ABB RobotStudio station: Proyecto_CesarGonzalez.rspag

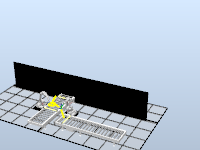
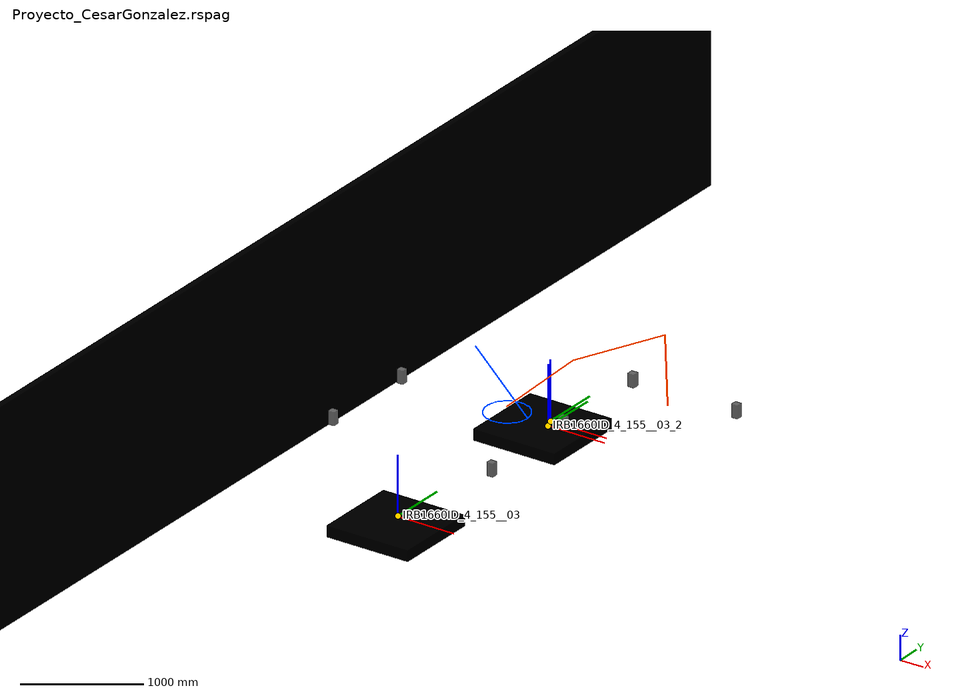
[picture v1: parts stored in the station drawn from their meshes, with robot base, taught points and paths (robot models come from the ABB library and are not in the file)]
--- station ---
Station Proyecto (saved by RobotStudio 21.2.9526.0)
Controller Controlador2, task T_ROB1: task frame (RAPID world) sits at (1630.73, 858.73, 94.26) mm in the station
Controller Controlador1, task T_ROB2: task frame (RAPID world) sits at (1633.69, -1291.95, 100) mm, rotated rx 0 ry 0 rz 90 deg in the station
Controller Controlador1, task T_ROB1: task frame (RAPID world) sits at (1633.69, -1291.95, 100) mm, rotated rx 0 ry 0 rz 90 deg in the station
Controller Controlador1
  mechanical unit ROB_1: IRB1660ID_4_155__03, 6 joints, base frame (0, 0, 0) mm
  mechanical unit ROB_2: IRB1660ID_4_155__03_2, 6 joints, base frame (0, 0, 0) mm
Controller Controlador2
  mechanical unit ROB_1: IRB1660ID_4_155__03_3, 6 joints, base frame (0, 0, 0) mm
Layout (positions relative to the parent item):
  - 950_4000_h2 [part, from Equipment\Conveyor 950 4000 h2.rslib] at (-254.72, -756.17, 0) mm
  - IRB1660ID_4_155__03 [mechanism, from Robots\IRB1660ID_4_155__03.rslib] at (1633.69, -1291.95, 100) mm, rotated rx 0 ry 0 rz 90 deg; joint values [-0.6056, 0.2499, 0.2095, 0.6847, 0.6619, -1.1198] (rad or m)
  - Pedestal1 [part] at (1259.57, -1762.3, 0) mm, size 800 x 800 x 100 mm
  - MyTool [mechanism, from Training Objects\myTool.rslib] at (2186.3, -401.7, 957.93) mm, rotated rx -179.96 ry 39.06 rz -86.55 deg
  - Cubo [part] at (3490.77, -286.76, 436.4) mm, size 400 x 400 x 300 mm
  - Tapa [part] at (2580.97, 4280.73, 447.22) mm, size 400 x 397.8 x 50 mm
  - 950_4000_h2_3 [part, from Equipment\Conveyor 950 4000 h2.rslib] at (3186.02, 749.76, 0) mm, rotated rx 0 ry 0 rz 90 deg
  - Pedestal2 [part] at (1208.56, 374.28, 0) mm, size 800 x 800 x 100 mm
  - IRB1660ID_4_155__03_2 [mechanism, from Robots\IRB1660ID_4_155__03.rslib] at (1674.65, 765.71, 100) mm; joint values [0, 0, 0, 0, 0.5236, 0] (rad or m)
  - PhysicsControl_cinta1 [smart component, from Components\PhysicsControl.rslib]
      properties: Object=cinta1; Behavior=1; SurfaceVelocity=0.2
  - PhysicsControl_cinta2 [smart component, from Components\PhysicsControl.rslib]
      properties: Object=cinta2; Behavior=1; SurfaceVelocity=0.2
  - Source_Cubo [smart component, from Components\Source.rslib]
      properties: Source=Cubo; Copy=(none); Parent=(none); Position=[3.49 -0.286 0.436]; Orientation=[0 0 0]; Transient=true; PhysicsBehavior=3
  - Source_Tapa [smart component, from Components\Source.rslib]
      properties: Source=Tapa; Copy=(none); Parent=(none); Position=[2.68 4.28 0.487]; Orientation=[0 0 0]; Transient=true; PhysicsBehavior=3
  - Pieza_2 [part] at (600.26, 166.12, 428.71) mm, size 60 x 60 x 120 mm
  - Pieza_3 [part] at (598.1, -796.46, 441.5) mm, size 60 x 60 x 120 mm
  - LineSensor_tapa [smart component, from Components\LineSensor.rslib] at (0, 259.06, -11.33) mm
      properties: Start=[2.263156 0.947069 0.47]; End=[3.181577 0.953591 0.47]; Radius=0; SensedPart=(none); SensedPoint=[2.49121630859375 1.20774780273438 0.458671112060547]
    - _sensorPart_ [part], size 918.4 x 6.5 x 0 mm
  - Pieza_4 [part] at (3189.53, 1175.28, 439.43) mm, size 60 x 60 x 120 mm
  - Pieza_5 [part] at (2172.87, 1169.42, 434.14) mm, size 60 x 60 x 120 mm
  - LineSensor_pegamento [smart component, from Components\LineSensor.rslib]
      properties: Start=[2.212913 -0.75684 0.495656]; End=[2.208882 0.177208 0.496891]; Radius=0; SensedPart=(none); SensedPoint=[0 0 0]
    - _sensorPart_ [part], size 4 x 934 x 1.2 mm
  - Pieza_6 [part] at (2178.88, 187.93, 436.89) mm, size 60 x 60 x 120 mm
  - Pieza_7 [part] at (2182.91, -828.74, 435.66) mm, size 60 x 60 x 120 mm
  - LineSensor_final [smart component, from Components\LineSensor.rslib]
      properties: Start=[0.628097 -0.720379 0.5015]; End=[0.630264 0.156269 0.488715]; Radius=0; SensedPart=(none); SensedPoint=[0 0 0]
    - _sensorPart_ [part], size 2.2 x 876.6 x 12.8 mm
  - cinta2 [part] at (2230.42, 4806.6, 338.68) mm, rotated rx 0 ry 0 rz -89.73 deg, size 4000 x 910 x 80 mm
  - cinta1 [part] at (-131.25, -752.86, 358) mm, size 4000 x 910 x 80 mm
  - IRB1660ID_4_155__03_3 [mechanism, from Robots\IRB1660ID_4_155__03.rslib] at (1630.73, 858.73, 94.26) mm; joint values [0, 0, 0, 0, 0.5236, 0] (rad or m)
  - Attacher [smart component, from Components\Attacher.rslib]
      properties: Parent=MyTool_2; Flange=0; Child=(none); Mount=false; Offset=[0 0 0]; Orientation=[0 0 0]
  - Detacher [smart component, from Components\Detacher.rslib]
      properties: Child=(none); KeepPosition=true
  - MyTool_2 [mechanism, from Training Objects\myTool.rslib] at (2575.61, 858.73, 1323.26) mm, rotated rx -180 ry 60 rz -180 deg
  - SimulationEvents [smart component, from Components\SimulationEvents.rslib]
  - Pared [part] at (28.4, -4684.22, 0) mm, size 60 x 10000 x 2000 mm
Attachment: Pedestal1 is attached to IRB1660ID_4_155__03 / Base
Attachment: MyTool is attached to IRB1660ID_4_155__03 / Link6
Attachment: Pedestal2 is attached to IRB1660ID_4_155__03_2 / Base
Attachment: PhysicsControl_cinta2 is attached to 950_4000_h2
Attachment: MyTool_2 is attached to IRB1660ID_4_155__03_3 / Link6
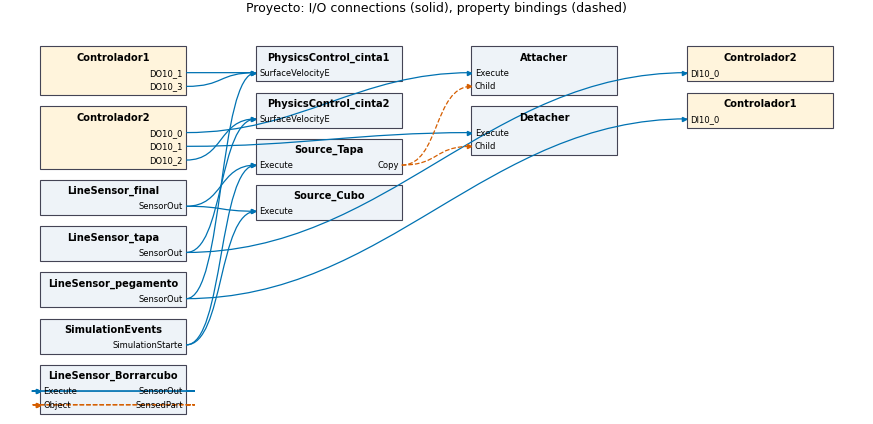
Station logic (signal -> signal, property => property):
  Controlador1.DO10_1 -> PhysicsControl_cinta1.SurfaceVelocityEnabled
  Controlador2.DO10_0 -> Attacher.Execute
  Controlador2.DO10_1 -> Detacher.Execute
  LineSensor_final.SensorOut -> Source_Tapa.Execute
  LineSensor_final.SensorOut -> Source_Cubo.Execute
  LineSensor_tapa.SensorOut -> PhysicsControl_cinta2.SurfaceVelocityEnabled
  LineSensor_pegamento.SensorOut -> PhysicsControl_cinta1.SurfaceVelocityEnabled
  LineSensor_pegamento.SensorOut -> Controlador1.DI10_0
  LineSensor_tapa.SensorOut -> Controlador2.DI10_0
  Controlador1.DO10_3 -> PhysicsControl_cinta1.SurfaceVelocityEnabled
  Controlador2.DO10_2 -> PhysicsControl_cinta2.SurfaceVelocityEnabled
  SimulationEvents.SimulationStarted -> Source_Tapa.Execute
  SimulationEvents.SimulationStarted -> Source_Cubo.Execute
  LineSensor_Borrarcubo.SensorOut -> Sink.Execute
  LineSensor_borrartapa.SensorOut -> Sink_3.Execute
  Source_Tapa.Copy => Detacher.Child
  Source_Tapa.Copy => Attacher.Child
  LineSensor_Borrarcubo.SensedPart => Sink.Object
  LineSensor_borrartapa.SensedPart => Sink_3.Object

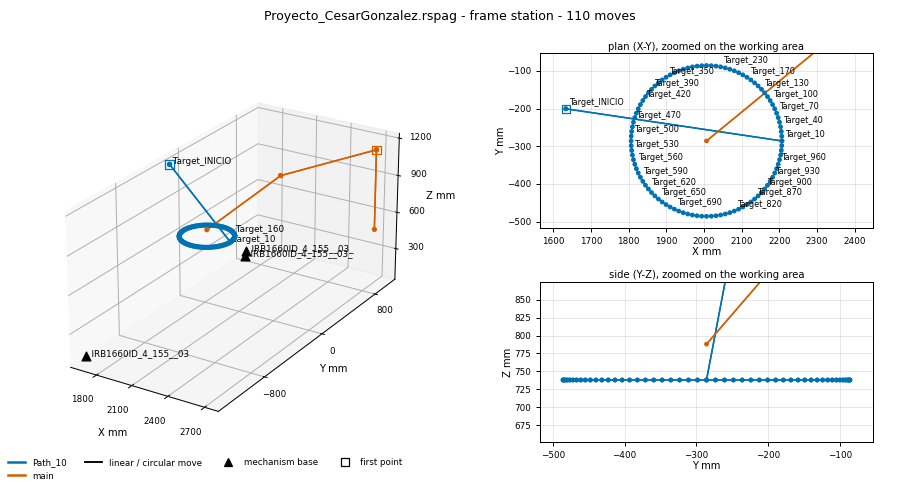
[picture p0: tool path of Proyecto_CesarGonzalez.rspag in frame station, 110 of 110 moves have a stored position in this frame; points joined in program order, loops and branches not executed]
--- Backups/Controlador1/RAPID/TASK1/PROGMOD/CalibData.mod ---
MODULE CalibData
    PERS tooldata MyTool:=[TRUE,[[31.7926,0,229.639],[0.945519,0,0.325568,0]],[1,[0,0,1],[1,0,0,0],0,0,0]];
ENDMODULE

--- Backups/Controlador1/RAPID/TASK1/PROGMOD/Module1.mod ---
MODULE Module1
    CONST robtarget Target_INICIO:=[[1091.194537048,0.000070456,1086.647618205],[0.190809199,-0.000000035,0.981627144,0.000000002],[0,-1,-1,0],[9E+09,9E+09,9E+09,9E+09,9E+09,9E+09]];
    CONST robtarget Target_10:=[[1005.945636056,-573.112362288,637.998901716],[0,-0.031410791,0.999506559,0],[0,0,0,0],[9E+09,9E+09,9E+09,9E+09,9E+09,9E+09]];
    CONST robtarget Target_20:=[[1018.503739937,-572.717707184,637.998901716],[0,-0.031410791,0.999506559,0],[0,0,0,0],[9E+09,9E+09,9E+09,9E+09,9E+09,9E+09]];
    CONST robtarget Target_30:=[[1031.01228267,-571.535300974,637.998901716],[0,-0.031410791,0.999506559,0],[0,0,0,0],[9E+09,9E+09,9E+09,9E+09,9E+09,9E+09]];
    CONST robtarget Target_40:=[[1043.421898751,-569.569810077,637.998901716],[0,-0.031410791,0.999506559,0],[0,0,0,0],[9E+09,9E+09,9E+09,9E+09,9E+09,9E+09]];
    CONST robtarget Target_50:=[[1055.683613094,-566.828991386,637.998901716],[0,-0.031410791,0.999506559,0],[0,0,0,0],[9E+09,9E+09,9E+09,9E+09,9E+09,9E+09]];
    CONST robtarget Target_60:=[[1067.749034316,-563.323661661,637.998901716],[0,-0.031410791,0.999506559,0],[0,0,0,0],[9E+09,9E+09,9E+09,9E+09,9E+09,9E+09]];
    CONST robtarget Target_70:=[[1079.57054571,-559.067654836,637.998901716],[0,-0.031410791,0.999506559,0],[0,0,0,0],[9E+09,9E+09,9E+09,9E+09,9E+09,9E+09]];
    CONST robtarget Target_80:=[[1091.101493172,-554.077767426,637.998901716],[0,-0.031410791,0.999506559,0],[0,0,0,0],[9E+09,9E+09,9E+09,9E+09,9E+09,9E+09]];
    CONST robtarget Target_90:=[[1102.296369321,-548.373692238,637.998901716],[0,-0.031410791,0.999506559,0],[0,0,0,0],[9E+09,9E+09,9E+09,9E+09,9E+09,9E+09]];
    CONST robtarget Target_100:=[[1113.110993094,-541.97794065,637.998901716],[0,-0.031410791,0.999506559,0],[0,0,0,0],[9E+09,9E+09,9E+09,9E+09,9E+09,9E+09]];
    CONST robtarget Target_110:=[[1123.502684113,-534.915753771,637.998901716],[0,-0.031410791,0.999506559,0],[0,0,0,0],[9E+09,9E+09,9E+09,9E+09,9E+09,9E+09]];
    CONST robtarget Target_120:=[[1133.43043112,-527.215002827,637.998901716],[0,-0.031410791,0.999506559,0],[0,0,0,0],[9E+09,9E+09,9E+09,9E+09,9E+09,9E+09]];
    CONST robtarget Target_130:=[[1142.855053833,-518.906079163,637.998901716],[0,-0.031410791,0.999506559,0],[0,0,0,0],[9E+09,9E+09,9E+09,9E+09,9E+09,9E+09]];
    CONST robtarget Target_140:=[[1151.739357573,-510.021774306,637.998901716],[0,-0.031410791,0.999506559,0],[0,0,0,0],[9E+09,9E+09,9E+09,9E+09,9E+09,9E+09]];
    CONST robtarget Target_150:=[[1160.048280052,-500.597150548,637.998901716],[0,-0.031410791,0.999506559,0],[0,0,0,0],[9E+09,9E+09,9E+09,9E+09,9E+09,9E+09]];
    CONST robtarget Target_160:=[[1167.749029747,-490.669402572,637.998901716],[0,-0.031410791,0.999506559,0],[0,0,0,0],[9E+09,9E+09,9E+09,9E+09,9E+09,9E+09]];
    CONST robtarget Target_170:=[[1174.811215319,-480.277710665,637.998901716],[0,-0.031410791,0.999506559,0],[0,0,0,0],[9E+09,9E+09,9E+09,9E+09,9E+09,9E+09]];
    CONST robtarget Target_180:=[[1181.206965548,-469.463086088,637.998901716],[0,-0.031410791,0.999506559,0],[0,0,0,0],[9E+09,9E+09,9E+09,9E+09,9E+09,9E+09]];
    CONST robtarget Target_190:=[[1186.911039328,-458.268209222,637.998901716],[0,-0.031410791,0.999506559,0],[0,0,0,0],[9E+09,9E+09,9E+09,9E+09,9E+09,9E+09]];
    CONST robtarget Target_200:=[[1191.900925287,-446.737261132,637.998901716],[0,-0.031410791,0.999506559,0],[0,0,0,0],[9E+09,9E+09,9E+09,9E+09,9E+09,9E+09]];
    CONST robtarget Target_210:=[[1196.156930626,-434.915749202,637.998901716],[0,-0.031410791,0.999506559,0],[0,0,0,0],[9E+09,9E+09,9E+09,9E+09,9E+09,9E+09]];
    CONST robtarget Target_220:=[[1199.662258834,-422.85032754,637.998901716],[0,-0.031410791,0.999506559,0],[0,0,0,0],[9E+09,9E+09,9E+09,9E+09,9E+09,9E+09]];
    CONST robtarget Target_230:=[[1202.403075983,-410.588612852,637.998901716],[0,-0.031410791,0.999506559,0],[0,0,0,0],[9E+09,9E+09,9E+09,9E+09,9E+09,9E+09]];
    CONST robtarget Target_240:=[[1204.368565319,-398.178996524,637.998901716],[0,-0.031410791,0.999506559,0],[0,0,0,0],[9E+09,9E+09,9E+09,9E+09,9E+09,9E+09]];
    CONST robtarget Target_250:=[[1205.550969956,-385.670453643,637.998901716],[0,-0.031410791,0.999506559,0],[0,0,0,0],[9E+09,9E+09,9E+09,9E+09,9E+09,9E+09]];
    CONST robtarget Target_260:=[[1205.94562348,-373.112349712,637.998901716],[0,-0.031410791,0.999506559,0],[0,0,0,0],[9E+09,9E+09,9E+09,9E+09,9E+09,9E+09]];
    CONST robtarget Target_270:=[[1205.550968376,-360.554245831,637.998901716],[0,-0.031410791,0.999506559,0],[0,0,0,0],[9E+09,9E+09,9E+09,9E+09,9E+09,9E+09]];
    CONST robtarget Target_280:=[[1204.368562167,-348.045703098,637.998901716],[0,-0.031410791,0.999506559,0],[0,0,0,0],[9E+09,9E+09,9E+09,9E+09,9E+09,9E+09]];
    CONST robtarget Target_290:=[[1202.40307127,-335.636087018,637.998901716],[0,-0.031410791,0.999506559,0],[0,0,0,0],[9E+09,9E+09,9E+09,9E+09,9E+09,9E+09]];
    CONST robtarget Target_300:=[[1199.662252579,-323.374372674,637.998901716],[0,-0.031410791,0.999506559,0],[0,0,0,0],[9E+09,9E+09,9E+09,9E+09,9E+09,9E+09]];
    CONST robtarget Target_310:=[[1196.156922853,-311.308951453,637.998901716],[0,-0.031410791,0.999506559,0],[0,0,0,0],[9E+09,9E+09,9E+09,9E+09,9E+09,9E+09]];
    CONST robtarget Target_320:=[[1191.900916029,-299.487440058,637.998901716],[0,-0.031410791,0.999506559,0],[0,0,0,0],[9E+09,9E+09,9E+09,9E+09,9E+09,9E+09]];
    CONST robtarget Target_330:=[[1186.911028619,-287.956492596,637.998901716],[0,-0.031410791,0.999506559,0],[0,0,0,0],[9E+09,9E+09,9E+09,9E+09,9E+09,9E+09]];
    CONST robtarget Target_340:=[[1181.206953431,-276.761616447,637.998901716],[0,-0.031410791,0.999506559,0],[0,0,0,0],[9E+09,9E+09,9E+09,9E+09,9E+09,9E+09]];
    CONST robtarget Target_350:=[[1174.811201842,-265.946992674,637.998901716],[0,-0.031410791,0.999506559,0],[0,0,0,0],[9E+09,9E+09,9E+09,9E+09,9E+09,9E+09]];
    CONST robtarget Target_360:=[[1167.749014963,-255.555301655,637.998901716],[0,-0.031410791,0.999506559,0],[0,0,0,0],[9E+09,9E+09,9E+09,9E+09,9E+09,9E+09]];
    CONST robtarget Target_370:=[[1160.048264019,-245.627554648,637.998901716],[0,-0.031410791,0.999506559,0],[0,0,0,0],[9E+09,9E+09,9E+09,9E+09,9E+09,9E+09]];
    CONST robtarget Target_380:=[[1151.739340356,-236.202931935,637.998901716],[0,-0.031410791,0.999506559,0],[0,0,0,0],[9E+09,9E+09,9E+09,9E+09,9E+09,9E+09]];
    CONST robtarget Target_390:=[[1142.855035499,-227.318628195,637.998901716],[0,-0.031410791,0.999506559,0],[0,0,0,0],[9E+09,9E+09,9E+09,9E+09,9E+09,9E+09]];
    CONST robtarget Target_400:=[[1133.43041174,-219.009705717,637.998901716],[0,-0.031410791,0.999506559,0],[0,0,0,0],[9E+09,9E+09,9E+09,9E+09,9E+09,9E+09]];
    CONST robtarget Target_410:=[[1123.502663765,-211.308956021,637.998901716],[0,-0.031410791,0.999506559,0],[0,0,0,0],[9E+09,9E+09,9E+09,9E+09,9E+09,9E+09]];
    CONST robtarget Target_420:=[[1113.110971858,-204.246770449,637.998901716],[0,-0.031410791,0.999506559,0],[0,0,0,0],[9E+09,9E+09,9E+09,9E+09,9E+09,9E+09]];
    CONST robtarget Target_430:=[[1102.29634728,-197.851020221,637.998901716],[0,-0.031410791,0.999506559,0],[0,0,0,0],[9E+09,9E+09,9E+09,9E+09,9E+09,9E+09]];
    CONST robtarget Target_440:=[[1091.101470414,-192.14694644,637.998901716],[0,-0.031410791,0.999506559,0],[0,0,0,0],[9E+09,9E+09,9E+09,9E+09,9E+09,9E+09]];
    CONST robtarget Target_450:=[[1079.570522325,-187.157060481,637.998901716],[0,-0.031410791,0.999506559,0],[0,0,0,0],[9E+09,9E+09,9E+09,9E+09,9E+09,9E+09]];
    CONST robtarget Target_460:=[[1067.749010395,-182.901055143,637.998901716],[0,-0.031410791,0.999506559,0],[0,0,0,0],[9E+09,9E+09,9E+09,9E+09,9E+09,9E+09]];
    CONST robtarget Target_470:=[[1055.683588733,-179.395726935,637.998901716],[0,-0.031410791,0.999506559,0],[0,0,0,0],[9E+09,9E+09,9E+09,9E+09,9E+09,9E+09]];
    CONST robtarget Target_480:=[[1043.421874044,-176.654909786,637.998901716],[0,-0.031410791,0.999506559,0],[0,0,0,0],[9E+09,9E+09,9E+09,9E+09,9E+09,9E+09]];
    CONST robtarget Target_490:=[[1031.012257717,-174.689420449,637.998901716],[0,-0.031410791,0.999506559,0],[0,0,0,0],[9E+09,9E+09,9E+09,9E+09,9E+09,9E+09]];
    CONST robtarget Target_500:=[[1018.503714835,-173.507015812,637.998901716],[0,-0.031410791,0.999506559,0],[0,0,0,0],[9E+09,9E+09,9E+09,9E+09,9E+09,9E+09]];
    CONST robtarget Target_510:=[[1005.945610905,-173.112362288,637.998901716],[0,-0.031410791,0.999506559,0],[0,0,0,0],[9E+09,9E+09,9E+09,9E+09,9E+09,9E+09]];
    CONST robtarget Target_520:=[[993.387507024,-173.507017392,637.998901716],[0,-0.031410791,0.999506559,0],[0,0,0,0],[9E+09,9E+09,9E+09,9E+09,9E+09,9E+09]];
    CONST robtarget Target_530:=[[980.878964291,-174.689423601,637.998901716],[0,-0.031410791,0.999506559,0],[0,0,0,0],[9E+09,9E+09,9E+09,9E+09,9E+09,9E+09]];
    CONST robtarget Target_540:=[[968.46934821,-176.654914498,637.998901716],[0,-0.031410791,0.999506559,0],[0,0,0,0],[9E+09,9E+09,9E+09,9E+09,9E+09,9E+09]];
    CONST robtarget Target_550:=[[956.207633867,-179.39573319,637.998901716],[0,-0.031410791,0.999506559,0],[0,0,0,0],[9E+09,9E+09,9E+09,9E+09,9E+09,9E+09]];
    CONST robtarget Target_560:=[[944.142212645,-182.901062915,637.998901716],[0,-0.031410791,0.999506559,0],[0,0,0,0],[9E+09,9E+09,9E+09,9E+09,9E+09,9E+09]];
    CONST robtarget Target_570:=[[932.320701251,-187.15706974,637.998901716],[0,-0.031410791,0.999506559,0],[0,0,0,0],[9E+09,9E+09,9E+09,9E+09,9E+09,9E+09]];
    CONST robtarget Target_580:=[[920.789753788,-192.146957149,637.998901716],[0,-0.031410791,0.999506559,0],[0,0,0,0],[9E+09,9E+09,9E+09,9E+09,9E+09,9E+09]];
    CONST robtarget Target_590:=[[909.59487764,-197.851032337,637.998901716],[0,-0.031410791,0.999506559,0],[0,0,0,0],[9E+09,9E+09,9E+09,9E+09,9E+09,9E+09]];
    CONST robtarget Target_600:=[[898.780253866,-204.246783926,637.998901716],[0,-0.031410791,0.999506559,0],[0,0,0,0],[9E+09,9E+09,9E+09,9E+09,9E+09,9E+09]];
    CONST robtarget Target_610:=[[888.388562848,-211.308970805,637.998901716],[0,-0.031410791,0.999506559,0],[0,0,0,0],[9E+09,9E+09,9E+09,9E+09,9E+09,9E+09]];
    CONST robtarget Target_620:=[[878.460815841,-219.009721749,637.998901716],[0,-0.031410791,0.999506559,0],[0,0,0,0],[9E+09,9E+09,9E+09,9E+09,9E+09,9E+09]];
    CONST robtarget Target_630:=[[869.036193127,-227.318645412,637.998901716],[0,-0.031410791,0.999506559,0],[0,0,0,0],[9E+09,9E+09,9E+09,9E+09,9E+09,9E+09]];
    CONST robtarget Target_640:=[[860.151889387,-236.202950269,637.998901716],[0,-0.031410791,0.999506559,0],[0,0,0,0],[9E+09,9E+09,9E+09,9E+09,9E+09,9E+09]];
    CONST robtarget Target_650:=[[851.842966909,-245.627574028,637.998901716],[0,-0.031410791,0.999506559,0],[0,0,0,0],[9E+09,9E+09,9E+09,9E+09,9E+09,9E+09]];
    CONST robtarget Target_660:=[[844.142217214,-255.555322003,637.998901716],[0,-0.031410791,0.999506559,0],[0,0,0,0],[9E+09,9E+09,9E+09,9E+09,9E+09,9E+09]];
    CONST robtarget Target_670:=[[837.080031642,-265.94701391,637.998901716],[0,-0.031410791,0.999506559,0],[0,0,0,0],[9E+09,9E+09,9E+09,9E+09,9E+09,9E+09]];
    CONST robtarget Target_680:=[[830.684281413,-276.761638488,637.998901716],[0,-0.031410791,0.999506559,0],[0,0,0,0],[9E+09,9E+09,9E+09,9E+09,9E+09,9E+09]];
    CONST robtarget Target_690:=[[824.980207633,-287.956515354,637.998901716],[0,-0.031410791,0.999506559,0],[0,0,0,0],[9E+09,9E+09,9E+09,9E+09,9E+09,9E+09]];
    CONST robtarget Target_700:=[[819.990321673,-299.487463443,637.998901716],[0,-0.031410791,0.999506559,0],[0,0,0,0],[9E+09,9E+09,9E+09,9E+09,9E+09,9E+09]];
    CONST robtarget Target_710:=[[815.734316335,-311.308975373,637.998901716],[0,-0.031410791,0.999506559,0],[0,0,0,0],[9E+09,9E+09,9E+09,9E+09,9E+09,9E+09]];
    CONST robtarget Target_720:=[[812.228988127,-323.374397035,637.998901716],[0,-0.031410791,0.999506559,0],[0,0,0,0],[9E+09,9E+09,9E+09,9E+09,9E+09,9E+09]];
    CONST robtarget Target_730:=[[809.488170978,-335.636111724,637.998901716],[0,-0.031410791,0.999506559,0],[0,0,0,0],[9E+09,9E+09,9E+09,9E+09,9E+09,9E+09]];
    CONST robtarget Target_740:=[[807.522681641,-348.045728052,637.998901716],[0,-0.031410791,0.999506559,0],[0,0,0,0],[9E+09,9E+09,9E+09,9E+09,9E+09,9E+09]];
    CONST robtarget Target_750:=[[806.340277005,-360.554270933,637.998901716],[0,-0.031410791,0.999506559,0],[0,0,0,0],[9E+09,9E+09,9E+09,9E+09,9E+09,9E+09]];
    CONST robtarget Target_760:=[[805.94562348,-373.112374864,637.998901716],[0,-0.031410791,0.999506559,0],[0,0,0,0],[9E+09,9E+09,9E+09,9E+09,9E+09,9E+09]];
    CONST robtarget Target_770:=[[806.340278584,-385.670478745,637.998901716],[0,-0.031410791,0.999506559,0],[0,0,0,0],[9E+09,9E+09,9E+09,9E+09,9E+09,9E+09]];
    CONST robtarget Target_780:=[[807.522684794,-398.179021477,637.998901716],[0,-0.031410791,0.999506559,0],[0,0,0,0],[9E+09,9E+09,9E+09,9E+09,9E+09,9E+09]];
    CONST robtarget Target_790:=[[809.488175691,-410.588637558,637.998901716],[0,-0.031410791,0.999506559,0],[0,0,0,0],[9E+09,9E+09,9E+09,9E+09,9E+09,9E+09]];
    CONST robtarget Target_800:=[[812.228994382,-422.850351901,637.998901716],[0,-0.031410791,0.999506559,0],[0,0,0,0],[9E+09,9E+09,9E+09,9E+09,9E+09,9E+09]];
    CONST robtarget Target_810:=[[815.734324107,-434.915773123,637.998901716],[0,-0.031410791,0.999506559,0],[0,0,0,0],[9E+09,9E+09,9E+09,9E+09,9E+09,9E+09]];
    CONST robtarget Target_820:=[[819.990330932,-446.737284517,637.998901716],[0,-0.031410791,0.999506559,0],[0,0,0,0],[9E+09,9E+09,9E+09,9E+09,9E+09,9E+09]];
    CONST robtarget Target_830:=[[824.980218342,-458.26823198,637.998901716],[0,-0.031410791,0.999506559,0],[0,0,0,0],[9E+09,9E+09,9E+09,9E+09,9E+09,9E+09]];
    CONST robtarget Target_840:=[[830.68429353,-469.463108128,637.998901716],[0,-0.031410791,0.999506559,0],[0,0,0,0],[9E+09,9E+09,9E+09,9E+09,9E+09,9E+09]];
    CONST robtarget Target_850:=[[837.080045118,-480.277731902,637.998901716],[0,-0.031410791,0.999506559,0],[0,0,0,0],[9E+09,9E+09,9E+09,9E+09,9E+09,9E+09]];
    CONST robtarget Target_860:=[[844.142231997,-490.66942292,637.998901716],[0,-0.031410791,0.999506559,0],[0,0,0,0],[9E+09,9E+09,9E+09,9E+09,9E+09,9E+09]];
    CONST robtarget Target_870:=[[851.842982941,-500.597169927,637.998901716],[0,-0.031410791,0.999506559,0],[0,0,0,0],[9E+09,9E+09,9E+09,9E+09,9E+09,9E+09]];
    CONST robtarget Target_880:=[[860.151906605,-510.021792641,637.998901716],[0,-0.031410791,0.999506559,0],[0,0,0,0],[9E+09,9E+09,9E+09,9E+09,9E+09,9E+09]];
    CONST robtarget Target_890:=[[869.036211462,-518.906096381,637.998901716],[0,-0.031410791,0.999506559,0],[0,0,0,0],[9E+09,9E+09,9E+09,9E+09,9E+09,9E+09]];
    CONST robtarget Target_900:=[[878.46083522,-527.215018859,637.998901716],[0,-0.031410791,0.999506559,0],[0,0,0,0],[9E+09,9E+09,9E+09,9E+09,9E+09,9E+09]];
    CONST robtarget Target_910:=[[888.388583196,-534.915768555,637.998901716],[0,-0.031410791,0.999506559,0],[0,0,0,0],[9E+09,9E+09,9E+09,9E+09,9E+09,9E+09]];
    CONST robtarget Target_920:=[[898.780275103,-541.977954127,637.998901716],[0,-0.031410791,0.999506559,0],[0,0,0,0],[9E+09,9E+09,9E+09,9E+09,9E+09,9E+09]];
    CONST robtarget Target_930:=[[909.59489968,-548.373704355,637.998901716],[0,-0.031410791,0.999506559,0],[0,0,0,0],[9E+09,9E+09,9E+09,9E+09,9E+09,9E+09]];
    CONST robtarget Target_940:=[[920.789776546,-554.077778135,637.998901716],[0,-0.031410791,0.999506559,0],[0,0,0,0],[9E+09,9E+09,9E+09,9E+09,9E+09,9E+09]];
    CONST robtarget Target_950:=[[932.320724636,-559.067664095,637.998901716],[0,-0.031410791,0.999506559,0],[0,0,0,0],[9E+09,9E+09,9E+09,9E+09,9E+09,9E+09]];
    CONST robtarget Target_960:=[[944.142236566,-563.323669433,637.998901716],[0,-0.031410791,0.999506559,0],[0,0,0,0],[9E+09,9E+09,9E+09,9E+09,9E+09,9E+09]];
    CONST robtarget Target_970:=[[956.207658228,-566.828997641,637.998901716],[0,-0.031410791,0.999506559,0],[0,0,0,0],[9E+09,9E+09,9E+09,9E+09,9E+09,9E+09]];
    CONST robtarget Target_980:=[[968.469372916,-569.56981479,637.998901716],[0,-0.031410791,0.999506559,0],[0,0,0,0],[9E+09,9E+09,9E+09,9E+09,9E+09,9E+09]];
    CONST robtarget Target_990:=[[980.878989244,-571.535304127,637.998901716],[0,-0.031410791,0.999506559,0],[0,0,0,0],[9E+09,9E+09,9E+09,9E+09,9E+09,9E+09]];
    CONST robtarget Target_1000:=[[993.387532125,-572.717708763,637.998901716],[0,-0.031410791,0.999506559,0],[0,0,0,0],[9E+09,9E+09,9E+09,9E+09,9E+09,9E+09]];
    CONST robtarget Target_1010:=[[1005.945636056,-573.112362288,637.998901716],[0,-0.031410791,0.999506559,0],[0,0,0,0],[9E+09,9E+09,9E+09,9E+09,9E+09,9E+09]];

    PROC Path_10()

        MoveL Target_INICIO,v1000,z100,MyTool\WObj:=wobj0;
        MoveL Target_10,v1000,z100,MyTool\WObj:=wobj0;
        MoveL Target_20,v1000,z100,MyTool\WObj:=wobj0;
        MoveL Target_30,v1000,z100,MyTool\WObj:=wobj0;
        MoveL Target_40,v1000,z100,MyTool\WObj:=wobj0;
        MoveL Target_50,v1000,z100,MyTool\WObj:=wobj0;
        MoveL Target_60,v1000,z100,MyTool\WObj:=wobj0;
        MoveL Target_70,v1000,z100,MyTool\WObj:=wobj0;
        MoveL Target_80,v1000,z100,MyTool\WObj:=wobj0;
        MoveL Target_90,v1000,z100,MyTool\WObj:=wobj0;
        MoveL Target_100,v1000,z100,MyTool\WObj:=wobj0;
        MoveL Target_110,v1000,z100,MyTool\WObj:=wobj0;
        MoveL Target_120,v1000,z100,MyTool\WObj:=wobj0;
        MoveL Target_130,v1000,z100,MyTool\WObj:=wobj0;
        MoveL Target_140,v1000,z100,MyTool\WObj:=wobj0;
        MoveL Target_150,v1000,z100,MyTool\WObj:=wobj0;
        MoveL Target_160,v1000,z100,MyTool\WObj:=wobj0;
        MoveL Target_170,v1000,z100,MyTool\WObj:=wobj0;
        MoveL Target_180,v1000,z100,MyTool\WObj:=wobj0;
        MoveL Target_190,v1000,z100,MyTool\WObj:=wobj0;
        MoveL Target_200,v1000,z100,MyTool\WObj:=wobj0;
        MoveL Target_210,v1000,z100,MyTool\WObj:=wobj0;
        MoveL Target_220,v1000,z100,MyTool\WObj:=wobj0;
        MoveL Target_230,v1000,z100,MyTool\WObj:=wobj0;
        MoveL Target_240,v1000,z100,MyTool\WObj:=wobj0;
        MoveL Target_250,v1000,z100,MyTool\WObj:=wobj0;
        MoveL Target_260,v1000,z100,MyTool\WObj:=wobj0;
        MoveL Target_270,v1000,z100,MyTool\WObj:=wobj0;
        MoveL Target_280,v1000,z100,MyTool\WObj:=wobj0;
        MoveL Target_290,v1000,z100,MyTool\WObj:=wobj0;
        MoveL Target_300,v1000,z100,MyTool\WObj:=wobj0;
        MoveL Target_310,v1000,z100,MyTool\WObj:=wobj0;
        MoveL Target_320,v1000,z100,MyTool\WObj:=wobj0;
        MoveL Target_330,v1000,z100,MyTool\WObj:=wobj0;
        MoveL Target_340,v1000,z100,MyTool\WObj:=wobj0;
        MoveL Target_350,v1000,z100,MyTool\WObj:=wobj0;
        MoveL Target_360,v1000,z100,MyTool\WObj:=wobj0;
        MoveL Target_370,v1000,z100,MyTool\WObj:=wobj0;
        MoveL Target_380,v1000,z100,MyTool\WObj:=wobj0;
        MoveL Target_390,v1000,z100,MyTool\WObj:=wobj0;
        MoveL Target_400,v1000,z100,MyTool\WObj:=wobj0;
        MoveL Target_410,v1000,z100,MyTool\WObj:=wobj0;
        MoveL Target_420,v1000,z100,MyTool\WObj:=wobj0;
        MoveL Target_430,v1000,z100,MyTool\WObj:=wobj0;
        MoveL Target_440,v1000,z100,MyTool\WObj:=wobj0;
        MoveL Target_450,v1000,z100,MyTool\WObj:=wobj0;
        MoveL Target_460,v1000,z100,MyTool\WObj:=wobj0;
        MoveL Target_470,v1000,z100,MyTool\WObj:=wobj0;
        MoveL Target_480,v1000,z100,MyTool\WObj:=wobj0;
        MoveL Target_490,v1000,z100,MyTool\WObj:=wobj0;
        MoveL Target_500,v1000,z100,MyTool\WObj:=wobj0;
        MoveL Target_510,v1000,z100,MyTool\WObj:=wobj0;
        MoveL Target_520,v1000,z100,MyTool\WObj:=wobj0;
        MoveL Target_530,v1000,z100,MyTool\WObj:=wobj0;
        MoveL Target_540,v1000,z100,MyTool\WObj:=wobj0;
        MoveL Target_550,v1000,z100,MyTool\WObj:=wobj0;
        MoveL Target_560,v1000,z100,MyTool\WObj:=wobj0;
        MoveL Target_570,v1000,z100,MyTool\WObj:=wobj0;
        MoveL Target_580,v1000,z100,MyTool\WObj:=wobj0;
        MoveL Target_590,v1000,z100,MyTool\WObj:=wobj0;
        MoveL Target_600,v1000,z100,MyTool\WObj:=wobj0;
        MoveL Target_610,v1000,z100,MyTool\WObj:=wobj0;
        MoveL Target_620,v1000,z100,MyTool\WObj:=wobj0;
        MoveL Target_630,v1000,z100,MyTool\WObj:=wobj0;
        MoveL Target_640,v1000,z100,MyTool\WObj:=wobj0;
        MoveL Target_650,v1000,z100,MyTool\WObj:=wobj0;
        MoveL Target_660,v1000,z100,MyTool\WObj:=wobj0;
        MoveL Target_670,v1000,z100,MyTool\WObj:=wobj0;
        MoveL Target_680,v1000,z100,MyTool\WObj:=wobj0;
        MoveL Target_690,v1000,z100,MyTool\WObj:=wobj0;
        MoveL Target_700,v1000,z100,MyTool\WObj:=wobj0;
        MoveL Target_710,v1000,z100,MyTool\WObj:=wobj0;
        MoveL Target_720,v1000,z100,MyTool\WObj:=wobj0;
        MoveL Target_730,v1000,z100,MyTool\WObj:=wobj0;
        MoveL Target_740,v1000,z100,MyTool\WObj:=wobj0;
        MoveL Target_750,v1000,z100,MyTool\WObj:=wobj0;
        MoveL Target_760,v1000,z100,MyTool\WObj:=wobj0;
        MoveL Target_770,v1000,z100,MyTool\WObj:=wobj0;
        MoveL Target_780,v1000,z100,MyTool\WObj:=wobj0;
        MoveL Target_790,v1000,z100,MyTool\WObj:=wobj0;
        MoveL Target_800,v1000,z100,MyTool\WObj:=wobj0;
        MoveL Target_810,v1000,z100,MyTool\WObj:=wobj0;
        MoveL Target_820,v1000,z100,MyTool\WObj:=wobj0;
        MoveL Target_830,v1000,z100,MyTool\WObj:=wobj0;
        MoveL Target_840,v1000,z100,MyTool\WObj:=wobj0;
        MoveL Target_850,v1000,z100,MyTool\WObj:=wobj0;
        MoveL Target_860,v1000,z100,MyTool\WObj:=wobj0;
        MoveL Target_870,v1000,z100,MyTool\WObj:=wobj0;
        MoveL Target_880,v1000,z100,MyTool\WObj:=wobj0;
        MoveL Target_890,v1000,z100,MyTool\WObj:=wobj0;
        MoveL Target_900,v1000,z100,MyTool\WObj:=wobj0;
        MoveL Target_910,v1000,z100,MyTool\WObj:=wobj0;
        MoveL Target_920,v1000,z100,MyTool\WObj:=wobj0;
        MoveL Target_930,v1000,z100,MyTool\WObj:=wobj0;
        MoveL Target_940,v1000,z100,MyTool\WObj:=wobj0;
        MoveL Target_950,v1000,z100,MyTool\WObj:=wobj0;
        MoveL Target_960,v1000,z100,MyTool\WObj:=wobj0;
        MoveL Target_970,v1000,z100,MyTool\WObj:=wobj0;
        MoveL Target_980,v1000,z100,MyTool\WObj:=wobj0;
        MoveL Target_990,v1000,z100,MyTool\WObj:=wobj0;
        MoveL Target_1000,v1000,z100,MyTool\WObj:=wobj0;
        MoveL Target_1010,v1000,z100,MyTool\WObj:=wobj0;
        MoveL Target_INICIO,v1000,z100,MyTool\WObj:=wobj0;
    ENDPROC

    PROC main()
        Reset DO10_1;
        Reset DO10_3;
        Set DO10_1;
      WAITDI DI10_0,1;
        Waittime 3;
        Path_10;
        WaitTime 20;
        Set DO10_3;
         WaitTime 10;

    ENDPROC
ENDMODULE

--- Backups/Controlador1/RAPID/TASK2/PROGMOD/CalibData.mod ---
MODULE CalibData
    PERS tooldata Ventosa:=[TRUE,[[0,0,130],[1,0,0,0]],[1,[0,0,1],[1,0,0,0],0,0,0]];
ENDMODULE

--- Backups/Controlador1/RAPID/TASK2/PROGMOD/RsTempModule.mod ---
MODULE RsTempModule
ENDMODULE

--- Backups/Controlador2/RAPID/TASK1/PROGMOD/CalibData.mod ---
MODULE CalibData
    PERS tooldata Ventosa:=[TRUE,[[0,0,130],[1,0,0,0]],[1,[0,0,1],[1,0,0,0],0,0,0]];
    PERS tooldata MyTool:=[TRUE,[[31.7926,0,229.639],[0.945519,0,0.325568,0]],[1,[0,0,1],[1,0,0,0],0,0,0]];
ENDMODULE

--- Backups/Controlador2/RAPID/TASK1/PROGMOD/Module1.mod ---
MODULE Module1
        CONST robtarget Target_INICIO:=[[1057.456732003,0,1164],[0.5,0,0.866025404,0],[0,-1,0,0],[9E+09,9E+09,9E+09,9E+09,9E+09,9E+09]];
    CONST robtarget Target_10:=[[1127.850265537,0,1086.64730631],[0.190808996,0,0.981627183,0],[0,-1,0,0],[9E+09,9E+09,9E+09,9E+09,9E+09,9E+09]];
    CONST robtarget Target_20:=[[525.913410499,-917.403850393,1164],[0.432628304,0.434163854,0.749334203,-0.250664618],[-1,0,0,0],[9E+09,9E+09,9E+09,9E+09,9E+09,9E+09]];
    CONST robtarget Target_30:=[[376.065812425,-1144.734628319,643.734872171],[1,0,0,0],[-1,0,0,3],[9E+09,9E+09,9E+09,9E+09,9E+09,9E+09]];
    CONST robtarget Target_60:=[[1049.265812425,147.665371681,374.417872171],[0.000000001,-0.000000001,1,0],[0,-2,1,0],[9E+09,9E+09,9E+09,9E+09,9E+09,9E+09]];
    CONST robtarget Target_40:=[[789.390514683,-805.548779902,1086.64730631],[0.1759124,0.380241374,0.904990842,-0.073911436],[-1,0,-1,0],[9E+09,9E+09,9E+09,9E+09,9E+09,9E+09]];
    CONST robtarget Target_50:=[[376.065812425,-1144.734628319,693.734872171],[0.000000001,0.382683431,0.923879533,0],[-1,0,-1,0],[9E+09,9E+09,9E+09,9E+09,9E+09,9E+09]];

    PROC main()
  Reset DO10_0;
    Reset DO10_1;
    Reset DO10_2;
    Set DO10_2;
    WaitDI DI10_0,1;
    WaitTime 0.5;
    MoveL Target_10,v500,fine,MyTool\WObj:=wobj0;
    MoveL Target_60,v500,fine,MyTool\WObj:=wobj0;
    WaitTime 1;
    Reset DO10_2;
    Set DO10_0;
    WaitTime 1;
     Reset DO10_0;
    MoveL Target_10,v500,fine,MyTool\WObj:=wobj0;
    MoveL Target_40,v500,fine,MyTool\WObj:=wobj0;
    MoveL Target_50,v500,fine,MyTool\WObj:=wobj0;
    WaitTime 1;
    Set DO10_1;
    MoveL Target_40,v500,fine,MyTool\WObj:=wobj0;
    MoveL Target_10,v500,fine,MyTool\WObj:=wobj0;
    Set DO10_2;
    WaitTime 1;

    ENDPROC


ENDMODULE

--- Backups/Controlador1/SYSPAR/EIO.cfg ---
EIO:CFG_1.0:6:1::
#
INDUSTRIAL_NETWORK:

      -Name "DeviceNet" -Label "DeviceNet Master/Slave Network" -Address "2"
#
DEVICENET_DEVICE:

      -Name "d653" -VendorName "ABB Robotics" -ProductName "Relay I/O Device"\
      -Label "DSQC 653 Relay I/O Device" -Address 10 -ProductCode 27\
      -DeviceType 7 -ConnectionType "COS" -OutputSize 1 -InputSize 1
#
DEVICENET_INTERNAL_DEVICE:

      -Name "DN_Internal_Device" -VendorName "ABB Robotics"\
      -ProductName "DeviceNet Internal Slave Device"
#
EIO_SIGNAL:

      -Name "DI10_0" -SignalType "DI" -Device "d653" -DeviceMap "0"

      -Name "DI10_1" -SignalType "DI" -Device "d653" -DeviceMap "1"

      -Name "DI10_2" -SignalType "DI" -Device "d653" -DeviceMap "2"

      -Name "DI10_3" -SignalType "DI" -Device "d653" -DeviceMap "3"

      -Name "DO10_0" -SignalType "DO" -Device "d653" -DeviceMap "0"

      -Name "DO10_1" -SignalType "DO" -Device "d653" -DeviceMap "1"

      -Name "DO10_2" -SignalType "DO" -Device "d653" -DeviceMap "2"

      -Name "DO10_3" -SignalType "DO" -Device "d653" -DeviceMap "3"

--- Backups/Controlador2/SYSPAR/EIO.cfg ---
EIO:CFG_1.0:6:1::
#
INDUSTRIAL_NETWORK:

      -Name "DeviceNet" -Label "DeviceNet Master/Slave Network" -Address "2"
#
DEVICENET_DEVICE:

      -Name "d652" -VendorName "ABB Robotics" -ProductName "24 VDC I/O Device"\
      -Label "DSQC 652 24 VDC I/O Device" -Address 10 -ProductCode 26\
      -DeviceType 7 -ConnectionType "COS" -OutputSize 2 -InputSize 2
#
DEVICENET_INTERNAL_DEVICE:

      -Name "DN_Internal_Device" -VendorName "ABB Robotics"\
      -ProductName "DeviceNet Internal Slave Device"
#
EIO_SIGNAL:

      -Name "DI10_0" -SignalType "DI" -Device "d652" -DeviceMap "0"

      -Name "DI10_1" -SignalType "DI" -Device "d652" -DeviceMap "1"

      -Name "DI10_2" -SignalType "DI" -Device "d652" -DeviceMap "2"

      -Name "DO10_0" -SignalType "DO" -Device "d652" -DeviceMap "0"

      -Name "DO10_1" -SignalType "DO" -Device "d652" -DeviceMap "1"

      -Name "DO10_2" -SignalType "DO" -Device "d652" -DeviceMap "2"

      -Name "DO10_3" -SignalType "DO" -Device "d652" -DeviceMap "3"
